TYPE HMI_DB_ADS :
STRUCT

	MANUAL				:REAL; (*Variables en provenance de la DB depuis le HMI*)
	AUTO				:REAL;
	NOT_AUS_RESET		:REAL;


END_STRUCT
END_TYPE

(* stored: Version 1.1.0.1, ProductVersion 3.1.0.26
   DUT HMI_DB_ADS: Id {eb69a4e0-789b-4840-84d2-2af0b067ab7e} *)
